PROGRAM MAIN
VAR
END_VAR

(*
 NAME:		16435-MOBILEHOIST
 CREATED:	10/30/2022 
 AUTHOR:	RRODRIGUEZ-HERNANDEZ
 FIRST PROTOTYPE
*)

DEADMANCONTROL();
ERROR_CASE_STATEMENT();
IOSTATE();
LIGHTLOGIC();
LOADINGLOGIC();
IO();

END_PROGRAM

(* stored: Version 1.1.0.1, ProductVersion 3.1.4024.11
   POU MAIN: Id {31c07508-205c-4447-851b-6a2075a38b4c}, SpecialFunc None *)
